{attribute addProperty BoxType "AX8640-0000-0029"}
{attribute addProperty Id "PSM_Controlword_for_axisAT %I*PSM_Controlword_for_axis_59B039C11620WcStateAT %I*WcState_98A4DF7520.250InfoDataAT %I*InfoData_0BDED7BF144180"}
{attribute addProperty CRC "4182654517"}
{attribute addProperty SizeInBites "162"}
{attribute addProperty SizeInBytes "20.25"}
TYPE AX8640_4A923142 :
STRUCT
	{attribute addProperty Name "PSM_Controlword_for_axis"}
	PSM_Controlword_for_axis : PSM_Controlword_for_axis_59B039C1;
	{attribute addProperty Name "WcState"}
	WcState : WcState_98A4DF75;
	{attribute addProperty Name "InfoData"}
	InfoData : InfoData_0BDED7BF;
END_STRUCT
END_TYPE

(* stored: Version 1.2.0.0, ProductVersion 3.1.4024.9
   DUT AX8640_4A923142: Id {ec561fc3-e729-45e4-8fb3-4d50089e7222} *)
